Universal Robots PolyScope program: urcap_test.urp

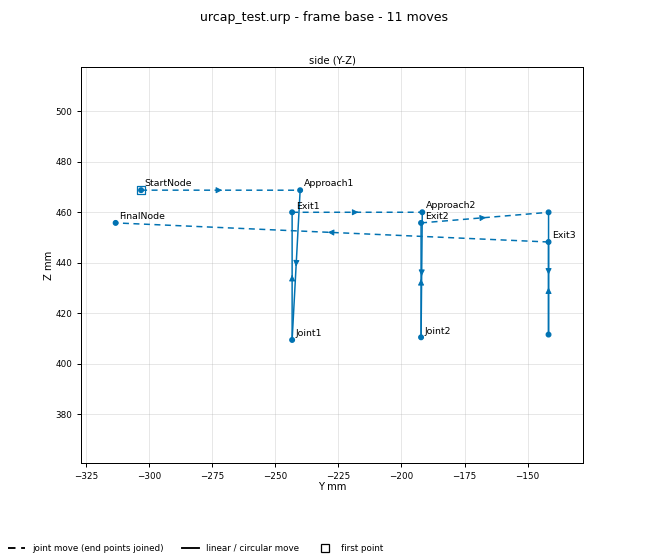
[picture p0: tool path of urcap_test.urp in frame base, 11 of 11 moves have a stored position in this frame; points joined in program order, loops and branches not executed]
Program urcap_test (installation=UPT directory=/programs/trial_codes createdIn=5.11.9.1010452 lastSavedIn=5.11.9.1010452 robotSerialNumber=20225580017)
Calibrated DH parameters: a=[0.000213, -0.129292, -0.392153, 0.000009, 0.000054, 0]; d=[0.162708, -398.929289, 399.773535, -0.710696, 0.099598, 0.099575]; alpha=[1.571486, 0.001015, 0.011079, 1.568772, -1.56976, 0]; deltaTheta=[0, -1.261618, 7.568654, -0.023852, -0.000001, 0]
Robot Program (runOnlyOnce=true)
  SafeHome (positionOptionType=SPEED_AND_ACCELERATION speed=1.047198 acceleration=1.396263 nextMotionTime=2)
  URCap UF Brazing Template (HeatControl, Ultraflex Power Technologies) dataModel(isExpanded=true, jointsNumber=3)
    'Starting Position'
    MoveJ speed 60 deg/s, acceleration 80 deg/s^2 (useActiveTCP=false) feature=Base
      Waypoint StartNode: TCP in base x=226.572 y=-303.083 z=468.66 mm, rx=2.1988 ry=2.2032 rz=-0.0006 rad; joints [-32.338, -70.597, -109.331, -88.521, 90.261, -212.606] deg
    Folder Joint 1
      'Approach Nodes'
      MoveJ speed 60 deg/s, acceleration 80 deg/s^2 (useActiveTCP=false) feature=Base
        Waypoint Approach1: TCP in base x=226.564 y=-240.097 z=468.633 mm, rx=2.1989 ry=2.2033 rz=-0.0007 rad; joints [-22.436, -63.025, -113.651, -91.87, 89.983, -202.75] deg
      'Joint Nodes'
      MoveL speed 40 mm/s, acceleration 100 mm/s^2 (useActiveTCP=false) feature=Base
        Waypoint Joint1: TCP in base x=227.686 y=-243.271 z=409.347 mm, rx=2.1988 ry=2.2031 rz=-0.0005 rad; joints [-22.947, -63.699, -121.979, -82.851, 89.997, -203.159] deg
        Set DigitalOutput pin=digital_out[2]; digitalValue=1
        Set DigitalOutput pin=config_out[2]; digitalValue=1
        URCap UF Brazing Node (HeatControl, Ultraflex Power Technologies) dataModel(powerport=0, onoffport=1, heatpowerdouble=80.0, heatdurationdouble=18.0)
        Waypoint Exit1: TCP in base x=227.658 y=-243.271 z=459.898 mm, rx=2.1989 ry=2.2031 rz=-0.0006 rad; joints [-22.921, -63.457, -114.71, -90.368, 89.997, -203.214] deg
    Folder Joint 2
      'Approach Nodes'
      MoveJ speed 60 deg/s, acceleration 80 deg/s^2 (useActiveTCP=false) feature=Base
        Waypoint Approach2: TCP in base x=224.91 y=-191.738 z=459.913 mm, rx=2.1989 ry=2.2032 rz=-0.0007 rad; joints [-13.065, -57.21, -117.564, -93.894, 89.736, -193.405] deg
      'Joint Nodes'
      MoveL speed 40 mm/s, acceleration 100 mm/s^2 (useActiveTCP=false) feature=Base
        Waypoint Joint2: TCP in base x=227.58 y=-192.218 z=410.388 mm, rx=2.199 ry=2.2032 rz=-0.0007 rad; joints [-13.068, -57.397, -124.728, -86.546, 89.74, -193.325] deg
        Set DigitalOutput pin=digital_out[2]; digitalValue=1
        Set DigitalOutput pin=config_out[2]; digitalValue=1
        URCap UF Brazing Node (HeatControl, Ultraflex Power Technologies) dataModel(powerport=0, onoffport=1, heatpowerdouble=80.0, heatdurationdouble=18.0)
        Waypoint Exit2: TCP in base x=227.6 y=-192.219 z=455.691 mm, rx=2.1989 ry=2.2031 rz=-0.0006 rad; joints [-13.04, -57.557, -118.04, -93.068, 89.74, -193.369] deg
    'Final Position'
    Folder Joint 3
      'Approach Nodes'
      MoveJ speed 60 deg/s, acceleration 80 deg/s^2 (useActiveTCP=false) feature=Base
        Waypoint Approach3: TCP in base x=224.915 y=-141.733 z=459.879 mm, rx=2.199 ry=2.2032 rz=-0.0008 rad; joints [-1.331, -52.063, -119.408, -97.411, 89.464, -181.714] deg
      'Joint Nodes'
      MoveL speed 40 mm/s, acceleration 100 mm/s^2 (useActiveTCP=false) feature=Base
        Waypoint Joint3: TCP in base x=227.506 y=-141.746 z=411.469 mm, rx=2.199 ry=2.2032 rz=-0.0008 rad; joints [-1.351, -51.767, -126.611, -90.503, 89.468, -181.656] deg
        Set DigitalOutput pin=digital_out[2]; digitalValue=1
        Set DigitalOutput pin=config_out[2]; digitalValue=1
        URCap UF Brazing Node (HeatControl, Ultraflex Power Technologies) dataModel(powerport=0, onoffport=0, heatpowerdouble=80.0, heatdurationdouble=18.0)
        Waypoint Exit3: TCP in base x=227.496 y=-141.747 z=448.132 mm, rx=2.1989 ry=2.2031 rz=-0.0007 rad; joints [-1.328, -52.208, -121.094, -95.573, 89.466, -181.688] deg
    MoveJ speed 60 deg/s, acceleration 80 deg/s^2 (useActiveTCP=false) feature=Base
      Waypoint FinalNode: TCP in base x=227.586 y=-313.157 z=455.692 mm, rx=2.1989 ry=2.2031 rz=-0.0006 rad; joints [-33.619, -71.962, -110.337, -86.142, 90.297, -213.854] deg
      SafeHome (positionOptionType=SPEED_AND_ACCELERATION speed=1.047198 acceleration=1.396263 nextMotionTime=2)
